% RSLogix 500 project LVD200820_BaseOnly_Mini.RSS, saved by version 11.00.00.00 %
PROJECT "LINL0619"    % processor: MicroLogix 1400 %

PROGRAM FILES
  LAD 2 "MAIN"  60 rungs  % Main Program Routine %
  LAD 4 "ENABLES"  16 rungs
  LAD 5 "FEED"  11 rungs  % normal %
  LAD 6 "SPEEDS"  12 rungs
  LAD 7 "HSC BOT"  5 rungs
  LAD 8 "HSC TOP"  5 rungs
  LAD 9 "1 MS STI"  22 rungs  % high speed %
  LAD 10 "SHIFT BOT"  8 rungs
  LAD 11 "SHIFT TOP"  10 rungs
  LAD 12 "BOTOPTIC"  3 rungs
  LAD 13 "BOTOPTMES"  7 rungs
  LAD 81 "I1"  1 rungs
  LAD 82 "I1 RESULT"  1 rungs
  LAD 83 "I1 PASS"  1 rungs
  LAD 84 "I1 FAIL"  1 rungs
  LAD 85 "I1 ACQ"  1 rungs
  LAD 86 "I1 TESTER"  1 rungs
  LAD 87 "I1 TRIG"  1 rungs
  LAD 88 "I1 FIFOSET"  1 rungs
  LAD 89 "I1 FIFOGET"  1 rungs
  LAD 90 "I1 DATA"  1 rungs
  LAD 91 "I1 FAULT"  1 rungs
  LAD 92 "I1 FIX1"  1 rungs
  LAD 93 "I1 FIX2"  1 rungs
  LAD 94 "I2"  1 rungs
  LAD 95 "I2 RESULT"  1 rungs
  LAD 96 "I2 PASS"  1 rungs
  LAD 97 "I2 FAIL"  1 rungs
  LAD 98 "I2 ACQ"  1 rungs
  LAD 99 "I2 TESTER"  1 rungs
  LAD 100 "I2 TRIG"  1 rungs
  LAD 101 "I2 FIFOSET"  1 rungs
  LAD 102 "I2 FIFOGET"  1 rungs
  LAD 103 "I2 DATA"  1 rungs
  LAD 104 "I2 FAULT"  1 rungs
  LAD 105 "I2 FIX1"  1 rungs
  LAD 106 "I2 FIX2"  1 rungs
  LAD 107 "I3"  1 rungs
  LAD 108 "I3 RESULT"  1 rungs
  LAD 109 "I3 PASS"  1 rungs
  LAD 110 "I3 FAIL"  1 rungs
  LAD 111 "I3 ACQ"  1 rungs
  LAD 112 "I3 TESTER"  1 rungs
  LAD 113 "I3 TRIG"  1 rungs
  LAD 114 "I3 FIFOSET"  1 rungs
  LAD 115 "I3 FIFOGET"  1 rungs
  LAD 116 "I3 DATA"  1 rungs
  LAD 117 "I3 FAULT"  1 rungs
  LAD 118 "I3 FIX1"  1 rungs
  LAD 119 "I3 FIX2"  1 rungs
  LAD 120 "I4"  1 rungs
  LAD 121 "I4 RESULT"  1 rungs
  LAD 122 "I4 PASS"  1 rungs
  LAD 123 "I4 FAIL"  1 rungs
  LAD 124 "I4 ACQ"  1 rungs
  LAD 125 "I4 TESTER"  1 rungs
  LAD 126 "I4 TRIG"  1 rungs
  LAD 127 "I4 FIFOSET"  1 rungs
  LAD 128 "I4 FIFOGET"  1 rungs
  LAD 129 "I4 DATA"  1 rungs
  LAD 130 "I4 FAULT"  1 rungs
  LAD 131 "I4 FIX1"  1 rungs
  LAD 132 "I4 FIX2"  1 rungs
  LAD 135 "XFER"  3 rungs
  LAD 137 "TOPOPTIC"  10 rungs
  LAD 138 "TOPOPVERT"  13 rungs
  LAD 139 "TOPOPREAL"  19 rungs
  LAD 140 "TOPOPTEST"  8 rungs
  LAD 141 "TOPOPRANGE"  6 rungs
  LAD 142 "TOPOPRANGE"  6 rungs
  LAD 143 "TOPOPOKAY"  6 rungs
  LAD 144 "TESTINJECT"  8 rungs
  LAD 148 "I5"  21 rungs
  LAD 149 "I5 RESULT"  7 rungs
  LAD 150 "I5 PASS"  6 rungs
  LAD 151 "I5 FAIL"  4 rungs
  LAD 152 "I5 ACQ"  9 rungs
  LAD 153 "I5 TESTER"  5 rungs
  LAD 154 "I5 TRIG"  5 rungs
  LAD 155 "I5 FIFOSET"  9 rungs
  LAD 156 "I5 FIFOGET"  8 rungs
  LAD 157 "I5 DATA"  3 rungs
  LAD 158 "I5 FAULT"  9 rungs
  LAD 159 "I5 FIX1"  5 rungs
  LAD 160 "I5 FIX2"  3 rungs
  LAD 161 "I6"  21 rungs
  LAD 162 "I6 RESULT"  7 rungs
  LAD 163 "I6 PASS"  5 rungs
  LAD 164 "I6 FAIL"  3 rungs
  LAD 165 "I6 ACQ"  8 rungs
  LAD 166 "I6 TESTER"  5 rungs
  LAD 167 "I6 TRIG"  5 rungs
  LAD 168 "I6 FIFOSET"  9 rungs
  LAD 169 "I6 FIFOGET"  8 rungs
  LAD 170 "I6 DATA"  3 rungs
  LAD 171 "I6 FAULT"  9 rungs
  LAD 172 "I6 FIX1"  5 rungs
  LAD 173 "I6 FIX2"  3 rungs
  LAD 174 "I7"  21 rungs
  LAD 175 "I7 RESULT"  7 rungs
  LAD 176 "I7 PASS"  6 rungs
  LAD 177 "I7 FAIL"  4 rungs
  LAD 178 "I7 ACQ"  9 rungs
  LAD 179 "I7 TESTER"  5 rungs
  LAD 180 "I7 TRIG"  5 rungs
  LAD 181 "I7 FIFOSET"  9 rungs
  LAD 182 "I7 FIFOGET"  8 rungs
  LAD 183 "I7 DATA"  3 rungs
  LAD 184 "I7 FAULT"  9 rungs
  LAD 185 "I7 FIX1"  5 rungs
  LAD 186 "I7 FIX2"  3 rungs
  LAD 187 "I8"  22 rungs
  LAD 188 "I8 RESULT"  7 rungs
  LAD 189 "I8 PASS"  6 rungs
  LAD 190 "I8 FAIL"  4 rungs
  LAD 191 "I8 ACQ"  9 rungs
  LAD 192 "I8 TESTER"  5 rungs
  LAD 193 "I8 TRIG"  5 rungs
  LAD 194 "I8 FIFOSET"  9 rungs
  LAD 195 "I8 FIFOGET"  8 rungs
  LAD 196 "I8 DATA"  3 rungs
  LAD 197 "I8 FAULT"  9 rungs
  LAD 198 "I8 FIX1"  5 rungs
  LAD 199 "I8 FIX2"  3 rungs
  LAD 200 "PASS BLOW"  15 rungs
  LAD 235 "TESTTRIGS"  7 rungs  % highspeed test triggers, not necessary %
  LAD 236 "TESTTRIG1"  4 rungs
  LAD 237 "TESTTRIG2"  4 rungs
  LAD 238 "TESTTRIG3"  4 rungs
  LAD 239 "TESTTRIG4"  4 rungs
  LAD 240 "TESTTRIG5"  4 rungs
  LAD 241 "TESTTRIG6"  4 rungs
  LAD 242 "TESTTRIG7"  4 rungs
  LAD 243 "TESTTRIG8"  4 rungs
  LAD 244 "PACKAGER"  28 rungs  % normal %
  LAD 245 "NO PACKAGE"  8 rungs
  LAD 246 "RATE1"  9 rungs
  LAD 247 "RATE2"  6 rungs
  LAD 248 "RESET RATE"  6 rungs
  LAD 249 "NP STOP"  8 rungs  % stop on no good %
  LAD 250 "SPEED BOT"  8 rungs  % high speed %
  LAD 251 "SPEED TOP"  8 rungs  % high speed %
  LAD 252 "P BOT"  7 rungs  % high speed %
  LAD 253 "P TOP"  7 rungs  % high speed %
  LAD 254 "TOTALCOUNT"  4 rungs
  LAD 255 "SAVED"  4 rungs

DATA FILES
  O0 OUTPUT  6 elements
  I1 INPUT  8 elements
  S2 STATUS  66 elements
  B3 BINARY  14 elements
  T4 TIMER  45 elements
  C5 COUNTER  1 elements
  R6 CONTROL  30 elements
  N7 INTEGER  200 elements
  F8 FLOAT  100 elements
  B12 HMI_BINARY  22 elements  % general use with hmi to avoid additional reads %
  L13  COUNTS  256 elements
  F14 HMI_FLOATS  100 elements
  N15 HMI_INTS  100 elements
  L16 HMI_LONGS  100 elements
  L19 RATE DATA  50 elements
  L20 I7TIMEFIFO  50 elements
  L21 I7POSFIFO  50 elements
  L22 I8TIMEFIFO  50 elements
  L23 I8POSFIFO  50 elements
  L30 INS5TIME  50 elements
  L31 INS5POS  50 elements
  L32 INS6TIME  50 elements
  L33 INS6POS  50 elements
  B34 BOT NG  128 elements
  B35 TOP NG  128 elements
  B36 BOTGOOD  128 elements
  B37 TOPGOOD1  128 elements
  B38 EX1 TEST  128 elements
  B39 TOPGOOD2  128 elements
  B40 EX2 TEST  128 elements
  N184 TEST INTS  50 elements
  L192 SPD OFFSET  50 elements
  B196 CTRL BITS  50 elements
  L199 USED  36 elements

LADDER 2 "MAIN"    % Main Program Routine %
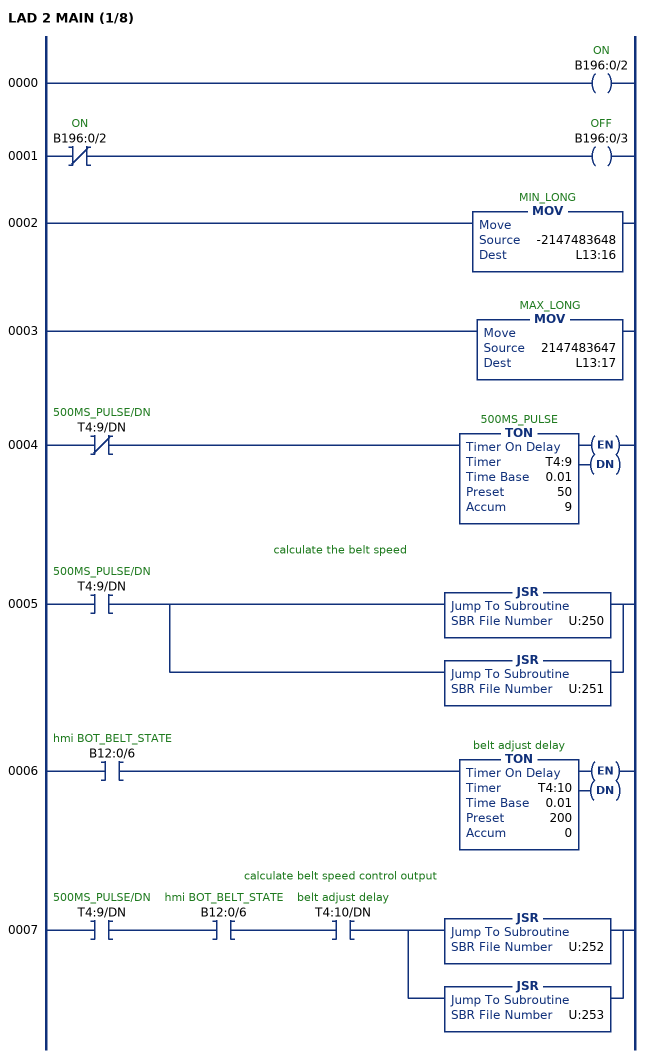
% Rung: 0 %
SOR OTE B196:0/2 EOR
%   B196:0/2  ON %
% Rung: 1 %
SOR XIO B196:0/2 OTE B196:0/3 EOR
%   B196:0/2  ON %
%   B196:0/3  OFF %
% Rung: 2 %
SOR MOV -2147483648 L13:16 EOR
%   L13:16  MIN_LONG %
% Rung: 3 %
SOR MOV 2147483647 L13:17 EOR
%   L13:17  MAX_LONG %
% Rung: 4 %
SOR XIO T4:9/DN TON T4:9 0.01 50 9 EOR
%   T4:9  500MS_PULSE %
% Rung: 5 %
% calculate the belt speed %
SOR XIC T4:9/DN BST JSR U:250 NXB JSR U:251 BND EOR
%   T4:9  500MS_PULSE %
% Rung: 6 %
SOR XIC B12:0/6 TON T4:10 0.01 200 0 EOR
%   B12:0/6  BOT_BELT_STATE  "hmi" %
%   T4:10  "belt adjust delay" %
% Rung: 7 %
% calculate belt speed control output %
SOR XIC T4:9/DN XIC B12:0/6 XIC T4:10/DN BST JSR U:252 NXB JSR U:253 BND EOR
%   T4:9  500MS_PULSE %
%   B12:0/6  BOT_BELT_STATE  "hmi" %
%   T4:10  "belt adjust delay" %

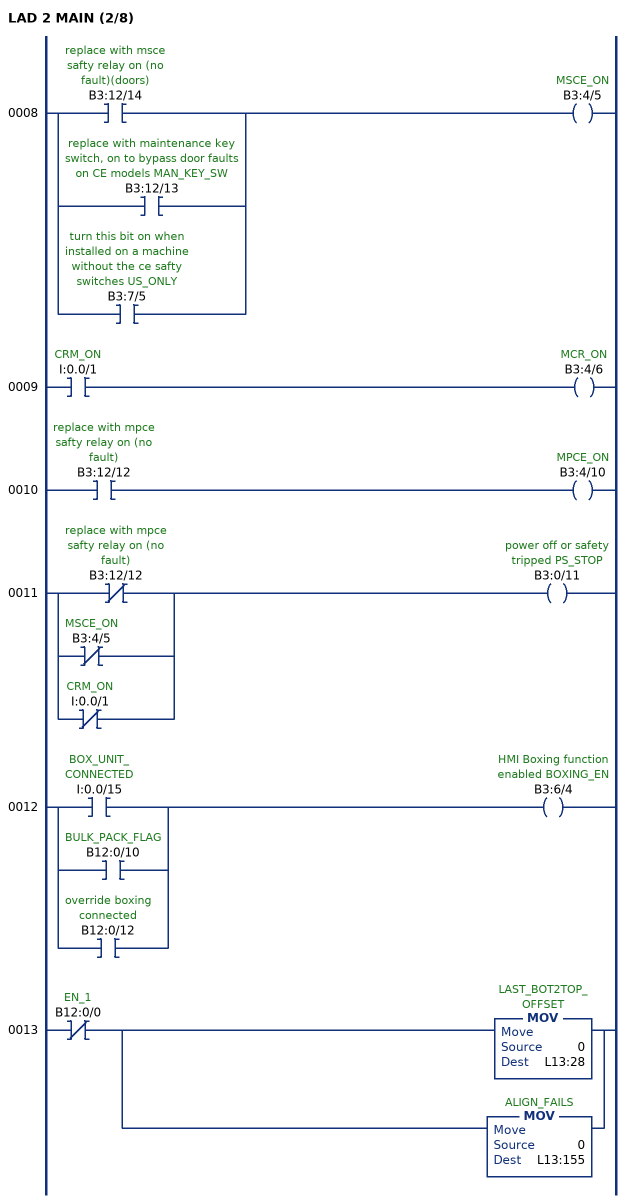
% Rung: 8 %
SOR BST XIC B3:12/14 NXB XIC B3:12/13 NXB XIC B3:7/5 BND OTE B3:4/5 EOR
%   B3:12/14  "replace with msce safty relay on (no fault)(doors)" %
%   B3:12/13  MAN_KEY_SW  "replace with maintenance key switch, on to bypass door faults on CE models" %
%   B3:7/5  US_ONLY  "turn this bit on when installed on a machine without the ce safty switches" %
%   B3:4/5  MSCE_ON %
% Rung: 9 %
SOR XIC I:0.0/1 OTE B3:4/6 EOR
%   I:0.0/1  CRM_ON %
%   B3:4/6  MCR_ON %
% Rung: 10 %
SOR XIC B3:12/12 OTE B3:4/10 EOR
%   B3:12/12  "replace with mpce safty relay on (no fault)" %
%   B3:4/10  MPCE_ON %
% Rung: 11 %
SOR BST XIO B3:12/12 NXB XIO B3:4/5 NXB XIO I:0.0/1 BND OTE B3:0/11 EOR
%   B3:12/12  "replace with mpce safty relay on (no fault)" %
%   B3:4/5  MSCE_ON %
%   I:0.0/1  CRM_ON %
%   B3:0/11  PS_STOP  "power off or safety tripped" %
% Rung: 12 %
SOR BST XIC I:0.0/15 NXB XIC B12:0/10 NXB XIC B12:0/12 BND OTE B3:6/4 EOR
%   I:0.0/15  BOX_UNIT_CONNECTED %
%   B12:0/10  BULK_PACK_FLAG %
%   B12:0/12  "override boxing connected" %
%   B3:6/4  BOXING_EN  "HMI Boxing function enabled" %
% Rung: 13 %
SOR XIO B12:0/0 BST MOV 0 L13:28 NXB MOV 0 L13:155 BND EOR
%   B12:0/0  EN_1 %
%   L13:28  LAST_BOT2TOP_OFFSET %
%   L13:155  ALIGN_FAILS %

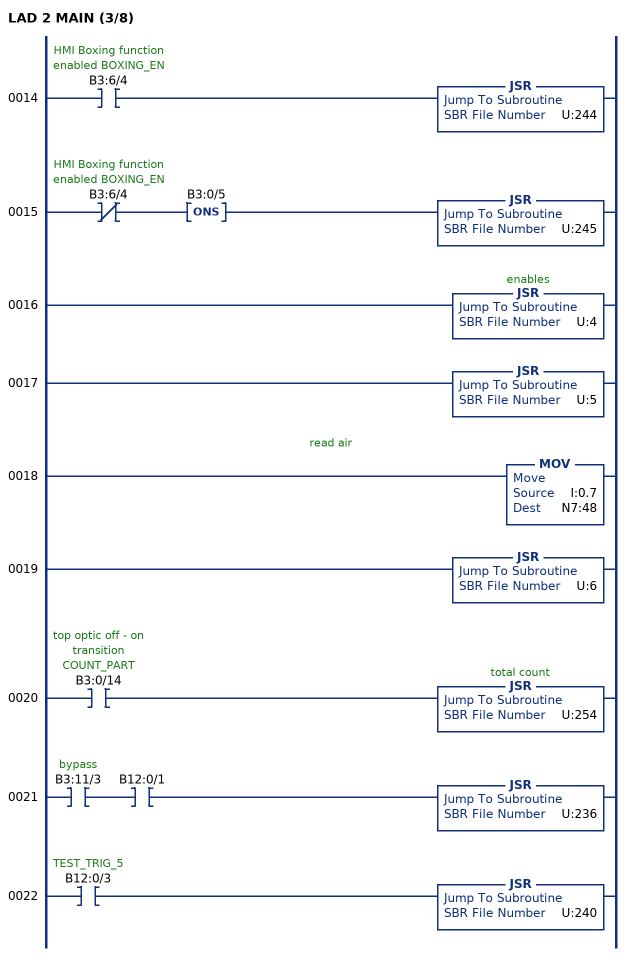
% Rung: 14 %
SOR XIC B3:6/4 JSR U:244 EOR
%   B3:6/4  BOXING_EN  "HMI Boxing function enabled" %
% Rung: 15 %
SOR XIO B3:6/4 ONS B3:0/5 JSR U:245 EOR
%   B3:6/4  BOXING_EN  "HMI Boxing function enabled" %
% Rung: 16 %
SOR JSR U:4 EOR
%   U:4  "enables" %
% Rung: 17 %
SOR JSR U:5 EOR
% Rung: 18 %
% read air %
SOR MOV I:0.7 N7:48 EOR
%   I:0.7  "Air Presure Sensor Input Signal" %
% Rung: 19 %
SOR JSR U:6 EOR
% Rung: 20 %
SOR XIC B3:0/14 JSR U:254 EOR
%   B3:0/14  COUNT_PART  "top optic off - on transition" %
%   U:254  "total count" %
% Rung: 21 %
SOR XIC B3:11/3 XIC B12:0/1 JSR U:236 EOR
%   B3:11/3  "bypass" %
% Rung: 22 %
SOR XIC B12:0/3 JSR U:240 EOR
%   B12:0/3  TEST_TRIG_5 %

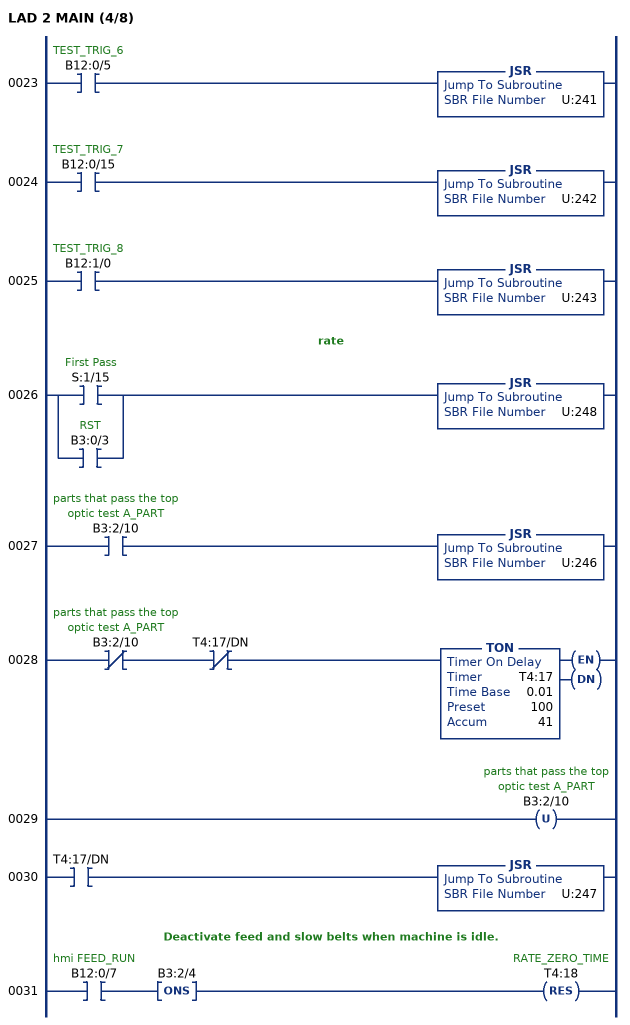
% Rung: 23 %
SOR XIC B12:0/5 JSR U:241 EOR
%   B12:0/5  TEST_TRIG_6 %
% Rung: 24 %
SOR XIC B12:0/15 JSR U:242 EOR
%   B12:0/15  TEST_TRIG_7 %
% Rung: 25 %
SOR XIC B12:1/0 JSR U:243 EOR
%   B12:1/0  TEST_TRIG_8 %
% Rung: 26 %
% TITLE: rate %
SOR BST XIC S:1/15 NXB XIC B3:0/3 BND JSR U:248 EOR
%   S:1/15  "First Pass" %
%   B3:0/3  RST %
% Rung: 27 %
SOR XIC B3:2/10 JSR U:246 EOR
%   B3:2/10  A_PART  "parts that pass the top optic test" %
% Rung: 28 %
SOR XIO B3:2/10 XIO T4:17/DN TON T4:17 0.01 100 41 EOR
%   B3:2/10  A_PART  "parts that pass the top optic test" %
% Rung: 29 %
SOR OTU B3:2/10 EOR
%   B3:2/10  A_PART  "parts that pass the top optic test" %
% Rung: 30 %
SOR XIC T4:17/DN JSR U:247 EOR
% Rung: 31 %
% TITLE: Deactivate feed and slow belts when machine is idle. %
SOR XIC B12:0/7 ONS B3:2/4 RES T4:18 EOR
%   B12:0/7  FEED_RUN  "hmi" %
%   T4:18  RATE_ZERO_TIME %

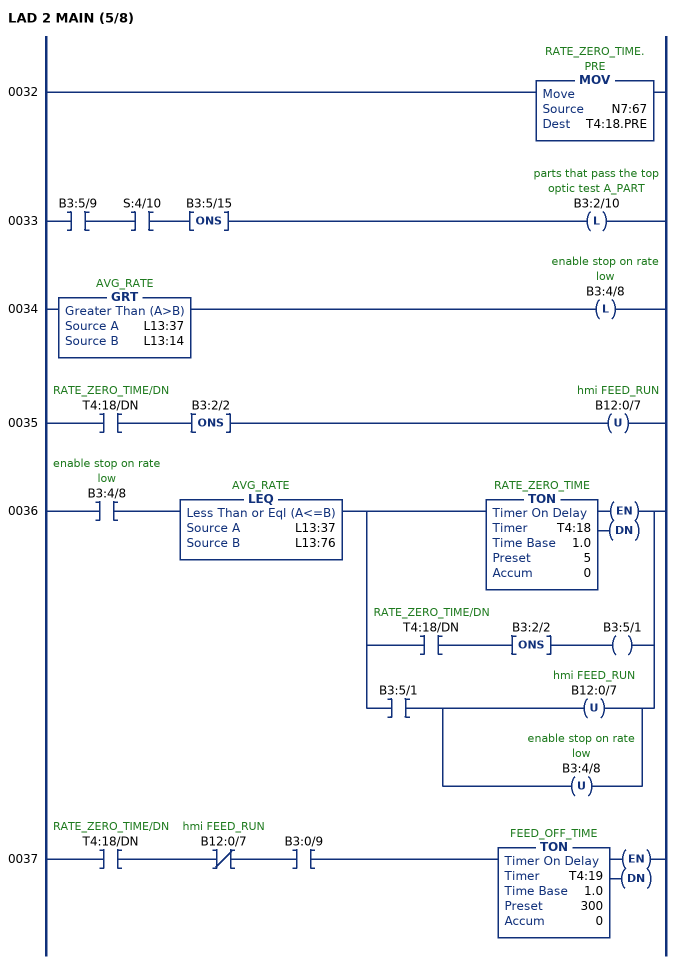
% Rung: 32 %
SOR MOV N7:67 T4:18.PRE EOR
%   N7:67  "empty bowl or jam bowl run time" %
%   T4:18  RATE_ZERO_TIME %
% Rung: 33 %
SOR XIC B3:5/9 XIC S:4/10 ONS B3:5/15 OTL B3:2/10 EOR
%   B3:2/10  A_PART  "parts that pass the top optic test" %
% Rung: 34 %
SOR GRT L13:37 L13:14 OTL B3:4/8 EOR
%   L13:37  AVG_RATE %
%   B3:4/8  "enable stop on rate low" %
% Rung: 35 %
SOR XIC T4:18/DN ONS B3:2/2 OTU B12:0/7 EOR
%   T4:18  RATE_ZERO_TIME %
%   B12:0/7  FEED_RUN  "hmi" %
% Rung: 36 %
SOR XIC B3:4/8 LEQ L13:37 L13:76 BST TON T4:18 1.0 5 0 NXB XIC T4:18/DN ONS B3:2/2 OTE B3:5/1 NXB XIC B3:5/1 BST OTU B12:0/7 NXB OTU B3:4/8 BND BND EOR
%   B3:4/8  "enable stop on rate low" %
%   L13:37  AVG_RATE %
%   T4:18  RATE_ZERO_TIME %
%   B12:0/7  FEED_RUN  "hmi" %
% Rung: 37 %
SOR XIC T4:18/DN XIO B12:0/7 XIC B3:0/9 TON T4:19 1.0 300 0 EOR
%   T4:18  RATE_ZERO_TIME %
%   B12:0/7  FEED_RUN  "hmi" %
%   T4:19  FEED_OFF_TIME %

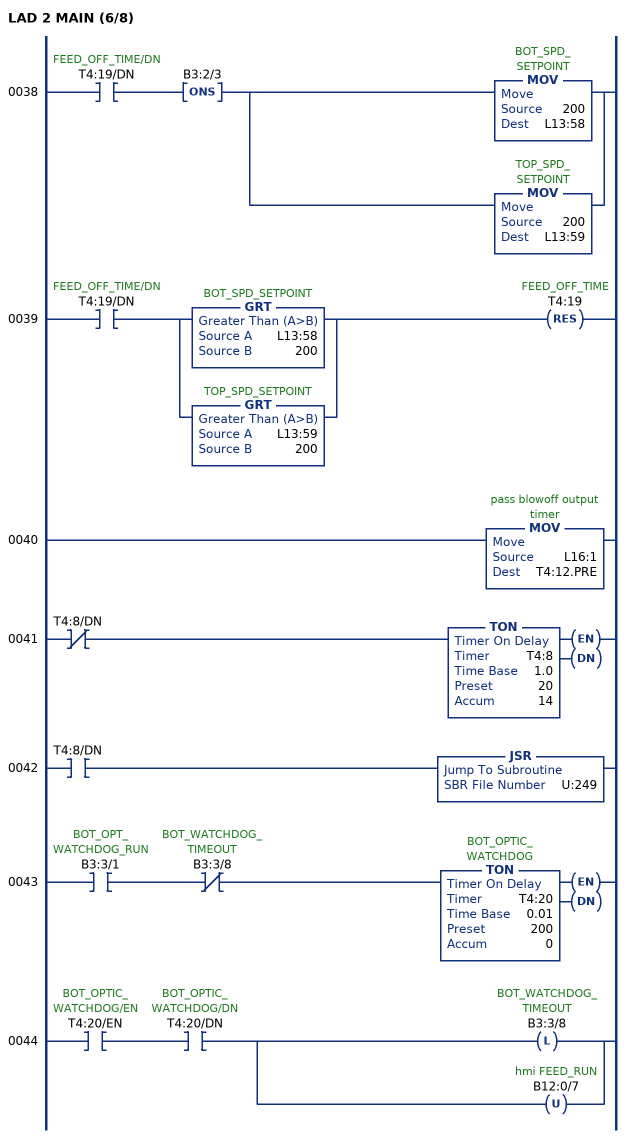
% Rung: 38 %
SOR XIC T4:19/DN ONS B3:2/3 BST MOV 200 L13:58 NXB MOV 200 L13:59 BND EOR
%   T4:19  FEED_OFF_TIME %
%   L13:58  BOT_SPD_SETPOINT %
%   L13:59  TOP_SPD_SETPOINT %
% Rung: 39 %
SOR XIC T4:19/DN BST GRT L13:58 200 NXB GRT L13:59 200 BND RES T4:19 EOR
%   T4:19  FEED_OFF_TIME %
%   L13:58  BOT_SPD_SETPOINT %
%   L13:59  TOP_SPD_SETPOINT %
% Rung: 40 %
SOR MOV L16:1 T4:12.PRE EOR
%   L16:1  BLOW_TIME %
%   T4:12  "pass blowoff output timer" %
% Rung: 41 %
SOR XIO T4:8/DN TON T4:8 1.0 20 14 EOR
% Rung: 42 %
SOR XIC T4:8/DN JSR U:249 EOR
% Rung: 43 %
SOR XIC B3:3/1 XIO B3:3/8 TON T4:20 0.01 200 0 EOR
%   B3:3/1  BOT_OPT_WATCHDOG_RUN %
%   B3:3/8  BOT_WATCHDOG_TIMEOUT %
%   T4:20  BOT_OPTIC_WATCHDOG %
% Rung: 44 %
SOR XIC T4:20/EN XIC T4:20/DN BST OTL B3:3/8 NXB OTU B12:0/7 BND EOR
%   T4:20  BOT_OPTIC_WATCHDOG %
%   B3:3/8  BOT_WATCHDOG_TIMEOUT %
%   B12:0/7  FEED_RUN  "hmi" %

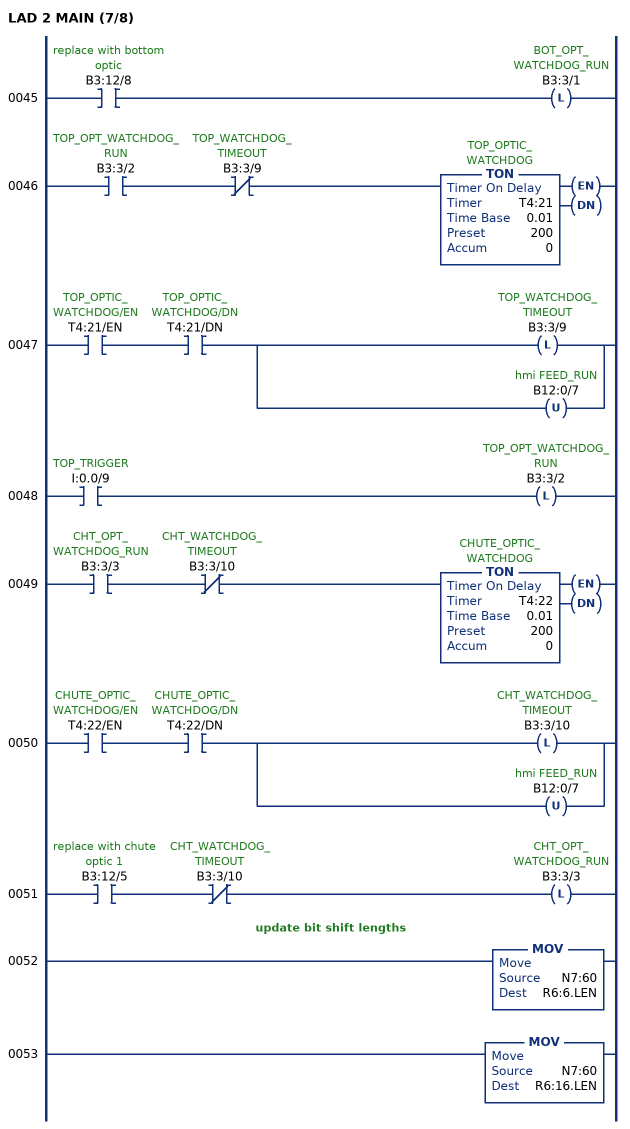
% Rung: 45 %
SOR XIC B3:12/8 OTL B3:3/1 EOR
%   B3:12/8  "replace with bottom optic" %
%   B3:3/1  BOT_OPT_WATCHDOG_RUN %
% Rung: 46 %
SOR XIC B3:3/2 XIO B3:3/9 TON T4:21 0.01 200 0 EOR
%   B3:3/2  TOP_OPT_WATCHDOG_RUN %
%   B3:3/9  TOP_WATCHDOG_TIMEOUT %
%   T4:21  TOP_OPTIC_WATCHDOG %
% Rung: 47 %
SOR XIC T4:21/EN XIC T4:21/DN BST OTL B3:3/9 NXB OTU B12:0/7 BND EOR
%   T4:21  TOP_OPTIC_WATCHDOG %
%   B3:3/9  TOP_WATCHDOG_TIMEOUT %
%   B12:0/7  FEED_RUN  "hmi" %
% Rung: 48 %
SOR XIC I:0.0/9 OTL B3:3/2 EOR
%   I:0.0/9  TOP_TRIGGER %
%   B3:3/2  TOP_OPT_WATCHDOG_RUN %
% Rung: 49 %
SOR XIC B3:3/3 XIO B3:3/10 TON T4:22 0.01 200 0 EOR
%   B3:3/3  CHT_OPT_WATCHDOG_RUN %
%   B3:3/10  CHT_WATCHDOG_TIMEOUT %
%   T4:22  CHUTE_OPTIC_WATCHDOG %
% Rung: 50 %
SOR XIC T4:22/EN XIC T4:22/DN BST OTL B3:3/10 NXB OTU B12:0/7 BND EOR
%   T4:22  CHUTE_OPTIC_WATCHDOG %
%   B3:3/10  CHT_WATCHDOG_TIMEOUT %
%   B12:0/7  FEED_RUN  "hmi" %
% Rung: 51 %
SOR XIC B3:12/5 XIO B3:3/10 OTL B3:3/3 EOR
%   B3:12/5  "replace with chute optic 1" %
%   B3:3/10  CHT_WATCHDOG_TIMEOUT %
%   B3:3/3  CHT_OPT_WATCHDOG_RUN %
% Rung: 52 %
% TITLE: update bit shift lengths %
SOR MOV N7:60 R6:6.LEN EOR
% Rung: 53 %
SOR MOV N7:60 R6:16.LEN EOR

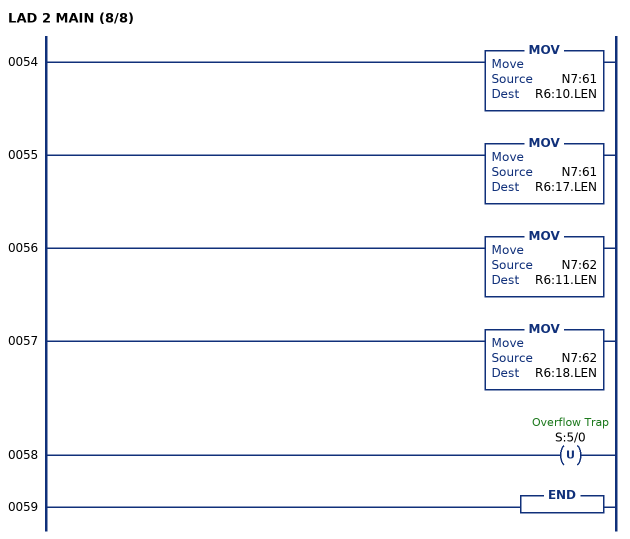
% Rung: 54 %
SOR MOV N7:61 R6:10.LEN EOR
% Rung: 55 %
SOR MOV N7:61 R6:17.LEN EOR
% Rung: 56 %
SOR MOV N7:62 R6:11.LEN EOR
% Rung: 57 %
SOR MOV N7:62 R6:18.LEN EOR
% Rung: 58 %
SOR OTU S:5/0 EOR
%   S:5/0  "Overflow Trap" %
% Rung: 59 %
SOR END EOR

LADDER 4 "ENABLES"
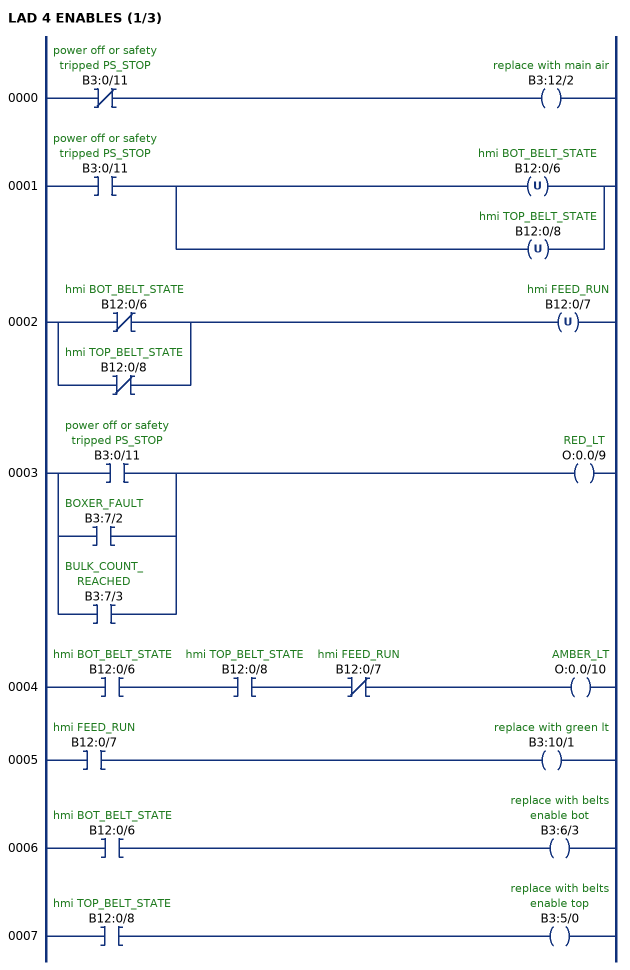
% Rung: 0 %
SOR XIO B3:0/11 OTE B3:12/2 EOR
%   B3:0/11  PS_STOP  "power off or safety tripped" %
%   B3:12/2  "replace with main air" %
% Rung: 1 %
SOR XIC B3:0/11 BST OTU B12:0/6 NXB OTU B12:0/8 BND EOR
%   B3:0/11  PS_STOP  "power off or safety tripped" %
%   B12:0/6  BOT_BELT_STATE  "hmi" %
%   B12:0/8  TOP_BELT_STATE  "hmi" %
% Rung: 2 %
SOR BST XIO B12:0/6 NXB XIO B12:0/8 BND OTU B12:0/7 EOR
%   B12:0/6  BOT_BELT_STATE  "hmi" %
%   B12:0/8  TOP_BELT_STATE  "hmi" %
%   B12:0/7  FEED_RUN  "hmi" %
% Rung: 3 %
SOR BST XIC B3:0/11 NXB XIC B3:7/2 NXB XIC B3:7/3 BND OTE O:0.0/9 EOR
%   B3:0/11  PS_STOP  "power off or safety tripped" %
%   B3:7/2  BOXER_FAULT %
%   B3:7/3  BULK_COUNT_REACHED %
%   O:0.0/9  RED_LT %
% Rung: 4 %
SOR XIC B12:0/6 XIC B12:0/8 XIO B12:0/7 OTE O:0.0/10 EOR
%   B12:0/6  BOT_BELT_STATE  "hmi" %
%   B12:0/8  TOP_BELT_STATE  "hmi" %
%   B12:0/7  FEED_RUN  "hmi" %
%   O:0.0/10  AMBER_LT %
% Rung: 5 %
SOR XIC B12:0/7 OTE B3:10/1 EOR
%   B12:0/7  FEED_RUN  "hmi" %
%   B3:10/1  "replace with green lt" %
% Rung: 6 %
SOR XIC B12:0/6 OTE B3:6/3 EOR
%   B12:0/6  BOT_BELT_STATE  "hmi" %
%   B3:6/3  "replace with belts enable bot" %
% Rung: 7 %
SOR XIC B12:0/8 OTE B3:5/0 EOR
%   B12:0/8  TOP_BELT_STATE  "hmi" %
%   B3:5/0  "replace with belts enable top" %

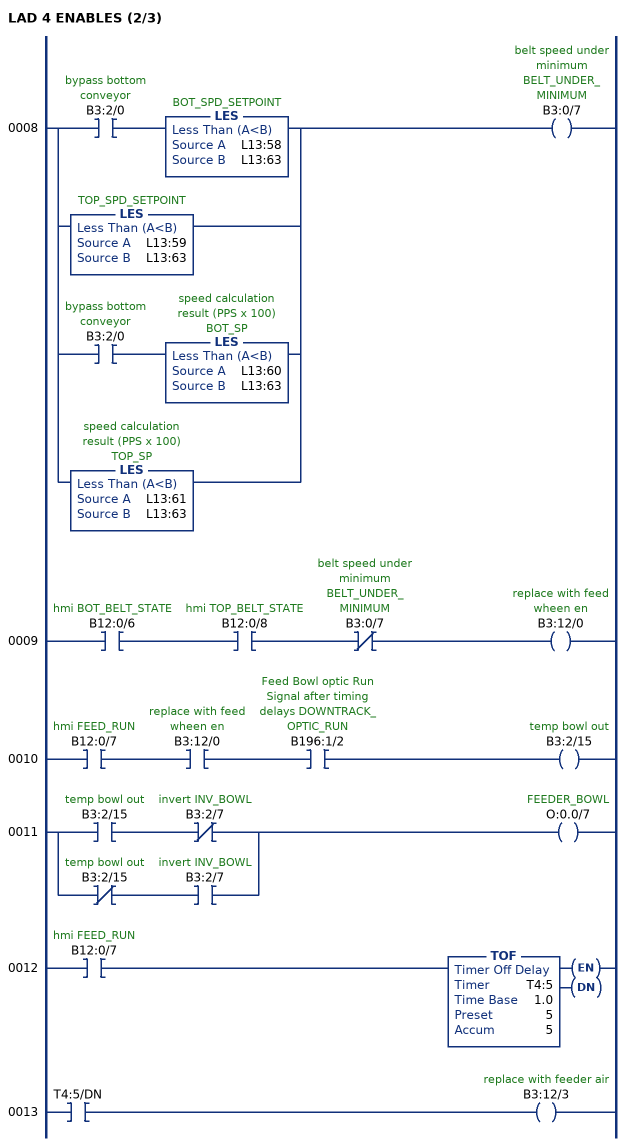
% Rung: 8 %
SOR BST XIC B3:2/0 LES L13:58 L13:63 NXB LES L13:59 L13:63 NXB XIC B3:2/0 LES L13:60 L13:63 NXB LES L13:61 L13:63 BND OTE B3:0/7 EOR
%   B3:2/0  "bypass bottom conveyor" %
%   L13:58  BOT_SPD_SETPOINT %
%   L13:63  "min belt speed" %
%   L13:59  TOP_SPD_SETPOINT %
%   L13:60  BOT_SP  "speed calculation result (PPS x 100)" %
%   L13:61  TOP_SP  "speed calculation result (PPS x 100)" %
%   B3:0/7  BELT_UNDER_MINIMUM  "belt speed under minimum" %
% Rung: 9 %
SOR XIC B12:0/6 XIC B12:0/8 XIO B3:0/7 OTE B3:12/0 EOR
%   B12:0/6  BOT_BELT_STATE  "hmi" %
%   B12:0/8  TOP_BELT_STATE  "hmi" %
%   B3:0/7  BELT_UNDER_MINIMUM  "belt speed under minimum" %
%   B3:12/0  "replace with feed wheen en" %
% Rung: 10 %
SOR XIC B12:0/7 XIC B3:12/0 XIC B196:1/2 OTE B3:2/15 EOR
%   B12:0/7  FEED_RUN  "hmi" %
%   B3:12/0  "replace with feed wheen en" %
%   B196:1/2  DOWNTRACK_OPTIC_RUN  "Feed Bowl optic Run Signal after timing delays" %
%   B3:2/15  "temp bowl out" %
% Rung: 11 %
SOR BST XIC B3:2/15 XIO B3:2/7 NXB XIO B3:2/15 XIC B3:2/7 BND OTE O:0.0/7 EOR
%   B3:2/15  "temp bowl out" %
%   B3:2/7  INV_BOWL  "invert" %
%   O:0.0/7  FEEDER_BOWL %
% Rung: 12 %
SOR XIC B12:0/7 TOF T4:5 1.0 5 5 EOR
%   B12:0/7  FEED_RUN  "hmi" %
% Rung: 13 %
SOR XIC T4:5/DN OTE B3:12/3 EOR
%   B3:12/3  "replace with feeder air" %

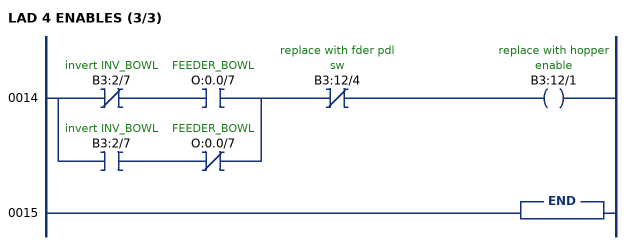
% Rung: 14 %
SOR BST XIO B3:2/7 XIC O:0.0/7 NXB XIC B3:2/7 XIO O:0.0/7 BND XIO B3:12/4 OTE B3:12/1 EOR
%   B3:2/7  INV_BOWL  "invert" %
%   O:0.0/7  FEEDER_BOWL %
%   B3:12/4  "replace with fder pdl sw" %
%   B3:12/1  "replace with hopper enable" %
% Rung: 15 %
SOR END EOR

LADDER 5 "FEED"    % normal %
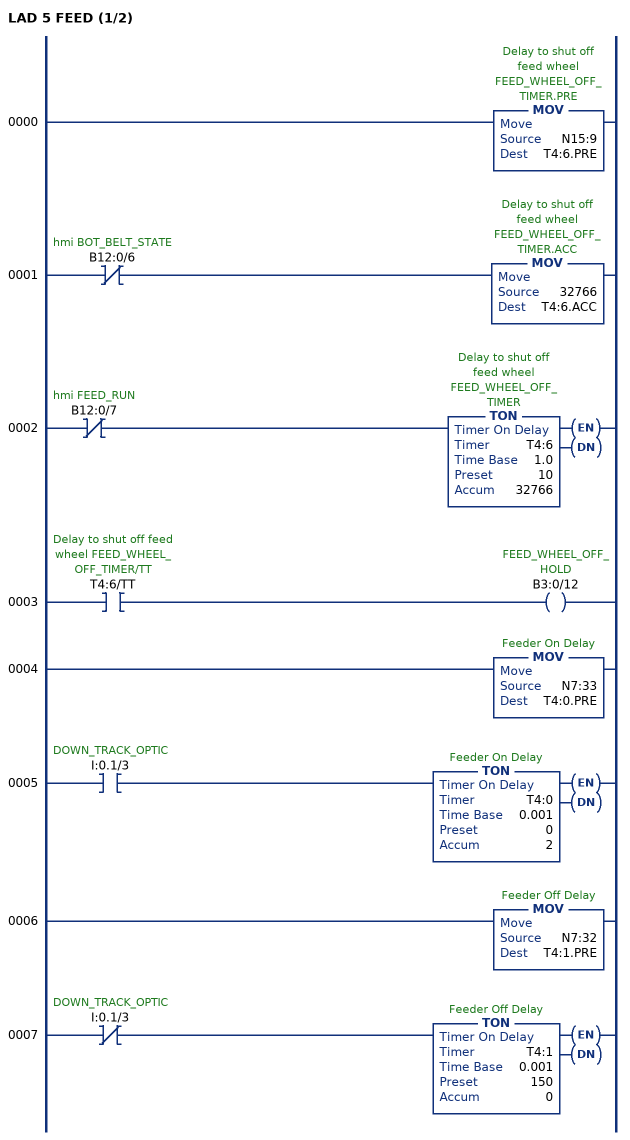
% Rung: 0 %
SOR MOV N15:9 T4:6.PRE EOR
%   N15:9  FEED_WHEEL_STOP_TIME %
%   T4:6  FEED_WHEEL_OFF_TIMER  "Delay to shut off feed wheel" %
% Rung: 1 %
SOR XIO B12:0/6 MOV 32766 T4:6.ACC EOR
%   B12:0/6  BOT_BELT_STATE  "hmi" %
%   T4:6  FEED_WHEEL_OFF_TIMER  "Delay to shut off feed wheel" %
% Rung: 2 %
SOR XIO B12:0/7 TON T4:6 1.0 10 32766 EOR
%   B12:0/7  FEED_RUN  "hmi" %
%   T4:6  FEED_WHEEL_OFF_TIMER  "Delay to shut off feed wheel" %
% Rung: 3 %
SOR XIC T4:6/TT OTE B3:0/12 EOR
%   T4:6  FEED_WHEEL_OFF_TIMER  "Delay to shut off feed wheel" %
%   B3:0/12  FEED_WHEEL_OFF_HOLD %
% Rung: 4 %
SOR MOV N7:33 T4:0.PRE EOR
%   N7:33  "down track on delay" %
%   T4:0  "Feeder On Delay" %
% Rung: 5 %
SOR XIC I:0.1/3 TON T4:0 0.001 0 2 EOR
%   I:0.1/3  DOWN_TRACK_OPTIC %
%   T4:0  "Feeder On Delay" %
% Rung: 6 %
SOR MOV N7:32 T4:1.PRE EOR
%   N7:32  "down track off delay" %
%   T4:1  "Feeder Off Delay" %
% Rung: 7 %
SOR XIO I:0.1/3 TON T4:1 0.001 150 0 EOR
%   I:0.1/3  DOWN_TRACK_OPTIC %
%   T4:1  "Feeder Off Delay" %

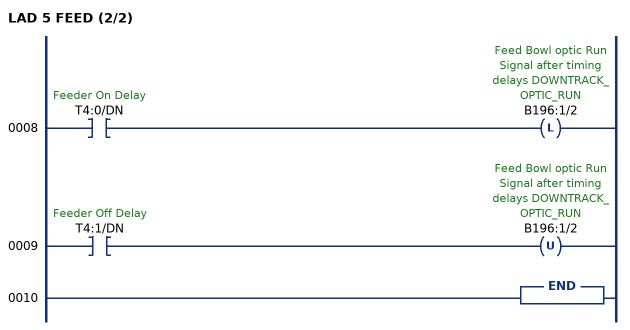
% Rung: 8 %
SOR XIC T4:0/DN OTL B196:1/2 EOR
%   T4:0  "Feeder On Delay" %
%   B196:1/2  DOWNTRACK_OPTIC_RUN  "Feed Bowl optic Run Signal after timing delays" %
% Rung: 9 %
SOR XIC T4:1/DN OTU B196:1/2 EOR
%   T4:1  "Feeder Off Delay" %
%   B196:1/2  DOWNTRACK_OPTIC_RUN  "Feed Bowl optic Run Signal after timing delays" %
% Rung: 10 %
SOR END EOR

LADDER 6 "SPEEDS"
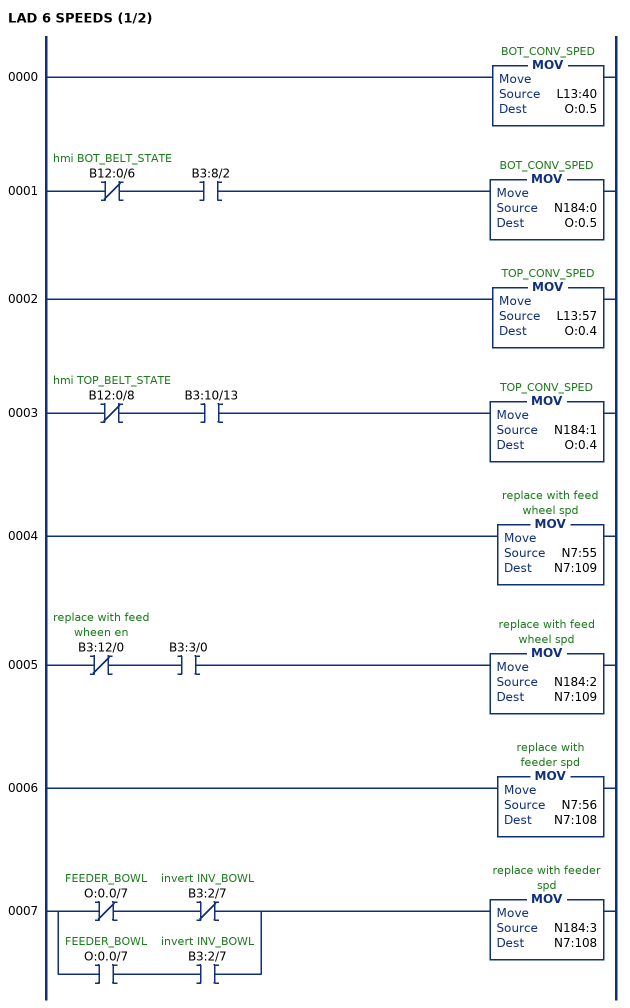
% Rung: 0 %
SOR MOV L13:40 O:0.5 EOR
%   L13:40  SCALED_BOT_VALUE %
%   O:0.5  BOT_CONV_SPED %
% Rung: 1 %
SOR XIO B12:0/6 XIC B3:8/2 MOV N184:0 O:0.5 EOR
%   B12:0/6  BOT_BELT_STATE  "hmi" %
%   O:0.5  BOT_CONV_SPED %
% Rung: 2 %
SOR MOV L13:57 O:0.4 EOR
%   L13:57  SCALED_TOP_VALUE %
%   O:0.4  TOP_CONV_SPED %
% Rung: 3 %
SOR XIO B12:0/8 XIC B3:10/13 MOV N184:1 O:0.4 EOR
%   B12:0/8  TOP_BELT_STATE  "hmi" %
%   O:0.4  TOP_CONV_SPED %
% Rung: 4 %
SOR MOV N7:55 N7:109 EOR
%   N7:109  "replace with feed wheel spd" %
% Rung: 5 %
SOR XIO B3:12/0 XIC B3:3/0 MOV N184:2 N7:109 EOR
%   B3:12/0  "replace with feed wheen en" %
%   N7:109  "replace with feed wheel spd" %
% Rung: 6 %
SOR MOV N7:56 N7:108 EOR
%   N7:108  "replace with feeder spd" %
% Rung: 7 %
SOR BST XIO O:0.0/7 XIO B3:2/7 NXB XIC O:0.0/7 XIC B3:2/7 BND MOV N184:3 N7:108 EOR
%   O:0.0/7  FEEDER_BOWL %
%   B3:2/7  INV_BOWL  "invert" %
%   N7:108  "replace with feeder spd" %

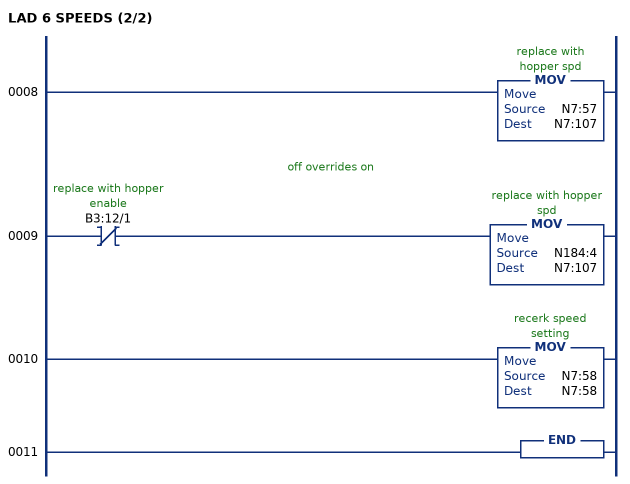
% Rung: 8 %
SOR MOV N7:57 N7:107 EOR
%   N7:107  "replace with hopper spd" %
% Rung: 9 %
% off overrides on %
SOR XIO B3:12/1 MOV N184:4 N7:107 EOR
%   B3:12/1  "replace with hopper enable" %
%   N7:107  "replace with hopper spd" %
% Rung: 10 %
SOR MOV N7:58 N7:58 EOR
%   N7:58  "recerk speed setting" %
% Rung: 11 %
SOR END EOR

LADDER 7 "HSC BOT"
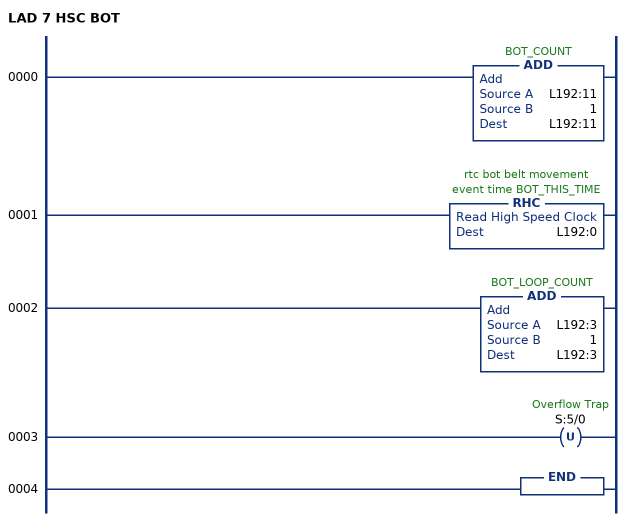
% Rung: 0 %
SOR ADD L192:11 1 L192:11 EOR
%   L192:11  BOT_COUNT %
% Rung: 1 %
SOR RHC L192:0 EOR
%   L192:0  BOT_THIS_TIME  "rtc bot belt movement event time" %
% Rung: 2 %
SOR ADD L192:3 1 L192:3 EOR
%   L192:3  BOT_LOOP_COUNT %
% Rung: 3 %
SOR OTU S:5/0 EOR
%   S:5/0  "Overflow Trap" %
% Rung: 4 %
SOR END EOR

LADDER 8 "HSC TOP"
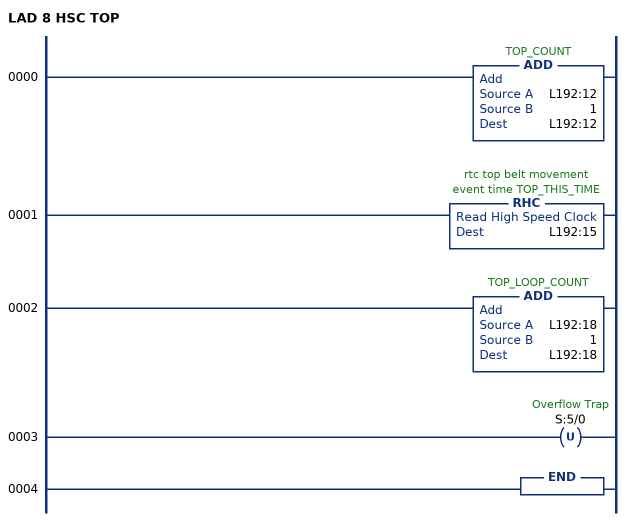
% Rung: 0 %
SOR ADD L192:12 1 L192:12 EOR
%   L192:12  TOP_COUNT %
% Rung: 1 %
SOR RHC L192:15 EOR
%   L192:15  TOP_THIS_TIME  "rtc top belt movement event time" %
% Rung: 2 %
SOR ADD L192:18 1 L192:18 EOR
%   L192:18  TOP_LOOP_COUNT %
% Rung: 3 %
SOR OTU S:5/0 EOR
%   S:5/0  "Overflow Trap" %
% Rung: 4 %
SOR END EOR

LADDER 9 "1 MS STI"    % high speed %
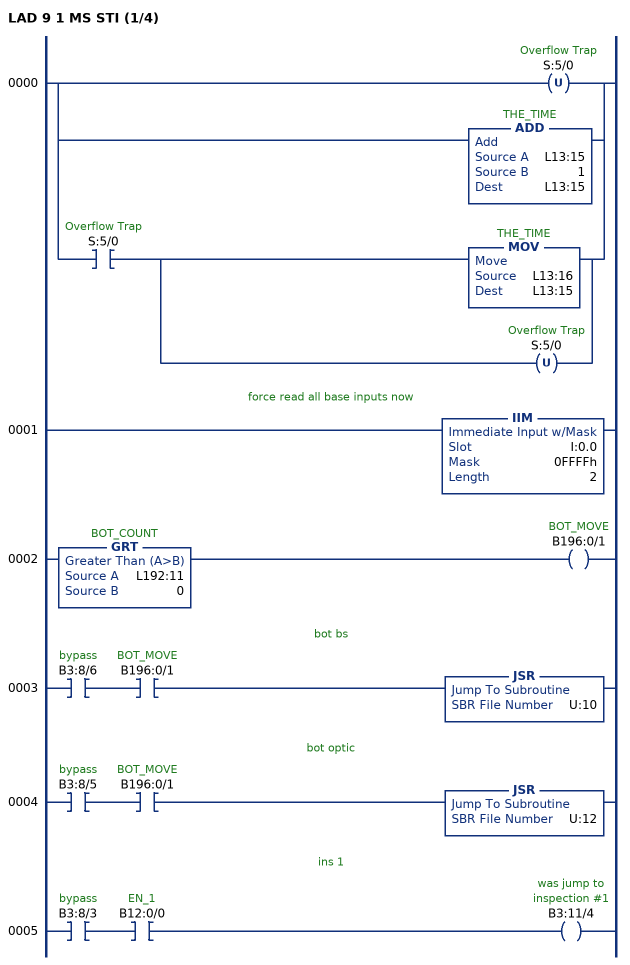
% Rung: 0 %
SOR BST OTU S:5/0 NXB ADD L13:15 1 L13:15 NXB XIC S:5/0 BST MOV L13:16 L13:15 NXB OTU S:5/0 BND BND EOR
%   S:5/0  "Overflow Trap" %
%   L13:15  THE_TIME %
%   L13:16  MIN_LONG %
% Rung: 1 %
% force read all base inputs now %
SOR IIM I:0.0 0FFFFh 2 EOR
% Rung: 2 %
SOR GRT L192:11 0 OTE B196:0/1 EOR
%   L192:11  BOT_COUNT %
%   B196:0/1  BOT_MOVE %
% Rung: 3 %
% bot bs %
SOR XIC B3:8/6 XIC B196:0/1 JSR U:10 EOR
%   B3:8/6  "bypass" %
%   B196:0/1  BOT_MOVE %
% Rung: 4 %
% bot optic %
SOR XIC B3:8/5 XIC B196:0/1 JSR U:12 EOR
%   B3:8/5  "bypass" %
%   B196:0/1  BOT_MOVE %
% Rung: 5 %
% ins 1 %
SOR XIC B3:8/3 XIC B12:0/0 OTE B3:11/4 EOR
%   B3:8/3  "bypass" %
%   B12:0/0  EN_1 %
%   B3:11/4  "was jump to inspection #1" %

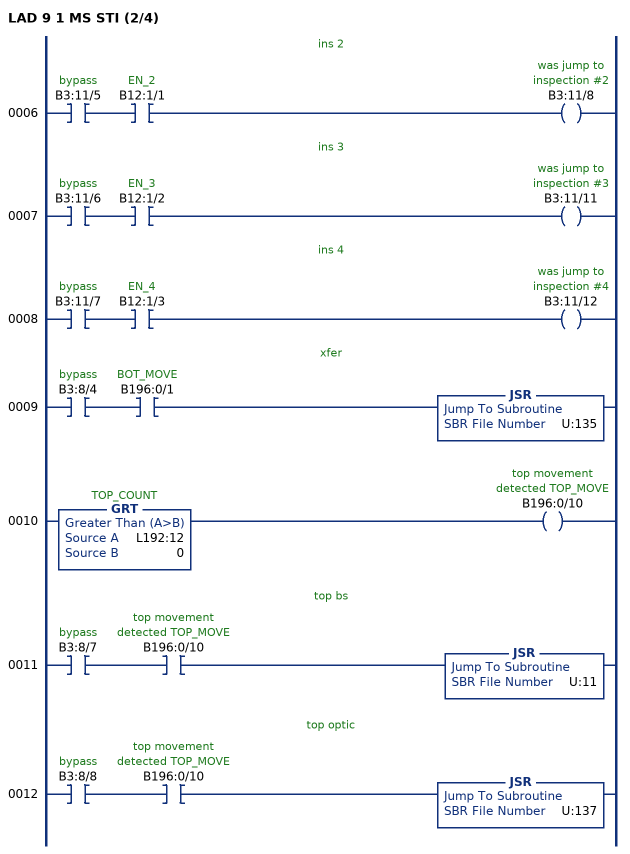
% Rung: 6 %
% ins 2 %
SOR XIC B3:11/5 XIC B12:1/1 OTE B3:11/8 EOR
%   B3:11/5  "bypass" %
%   B12:1/1  EN_2 %
%   B3:11/8  "was jump to inspection #2" %
% Rung: 7 %
% ins 3 %
SOR XIC B3:11/6 XIC B12:1/2 OTE B3:11/11 EOR
%   B3:11/6  "bypass" %
%   B12:1/2  EN_3 %
%   B3:11/11  "was jump to inspection #3" %
% Rung: 8 %
% ins 4 %
SOR XIC B3:11/7 XIC B12:1/3 OTE B3:11/12 EOR
%   B3:11/7  "bypass" %
%   B12:1/3  EN_4 %
%   B3:11/12  "was jump to inspection #4" %
% Rung: 9 %
% xfer %
SOR XIC B3:8/4 XIC B196:0/1 JSR U:135 EOR
%   B3:8/4  "bypass" %
%   B196:0/1  BOT_MOVE %
% Rung: 10 %
SOR GRT L192:12 0 OTE B196:0/10 EOR
%   L192:12  TOP_COUNT %
%   B196:0/10  TOP_MOVE  "top movement detected" %
% Rung: 11 %
% top bs %
SOR XIC B3:8/7 XIC B196:0/10 JSR U:11 EOR
%   B3:8/7  "bypass" %
%   B196:0/10  TOP_MOVE  "top movement detected" %
% Rung: 12 %
% top optic %
SOR XIC B3:8/8 XIC B196:0/10 JSR U:137 EOR
%   B3:8/8  "bypass" %
%   B196:0/10  TOP_MOVE  "top movement detected" %

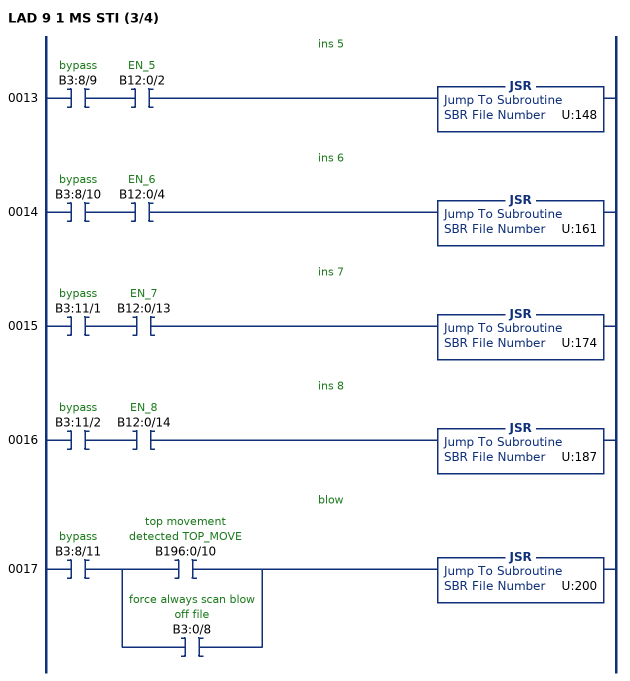
% Rung: 13 %
% ins 5 %
SOR XIC B3:8/9 XIC B12:0/2 JSR U:148 EOR
%   B3:8/9  "bypass" %
%   B12:0/2  EN_5 %
% Rung: 14 %
% ins 6 %
SOR XIC B3:8/10 XIC B12:0/4 JSR U:161 EOR
%   B3:8/10  "bypass" %
%   B12:0/4  EN_6 %
% Rung: 15 %
% ins 7 %
SOR XIC B3:11/1 XIC B12:0/13 JSR U:174 EOR
%   B3:11/1  "bypass" %
%   B12:0/13  EN_7 %
% Rung: 16 %
% ins 8 %
SOR XIC B3:11/2 XIC B12:0/14 JSR U:187 EOR
%   B3:11/2  "bypass" %
%   B12:0/14  EN_8 %
% Rung: 17 %
% blow %
SOR XIC B3:8/11 BST XIC B196:0/10 NXB XIC B3:0/8 BND JSR U:200 EOR
%   B3:8/11  "bypass" %
%   B196:0/10  TOP_MOVE  "top movement detected" %
%   B3:0/8  "force always scan blow off file" %

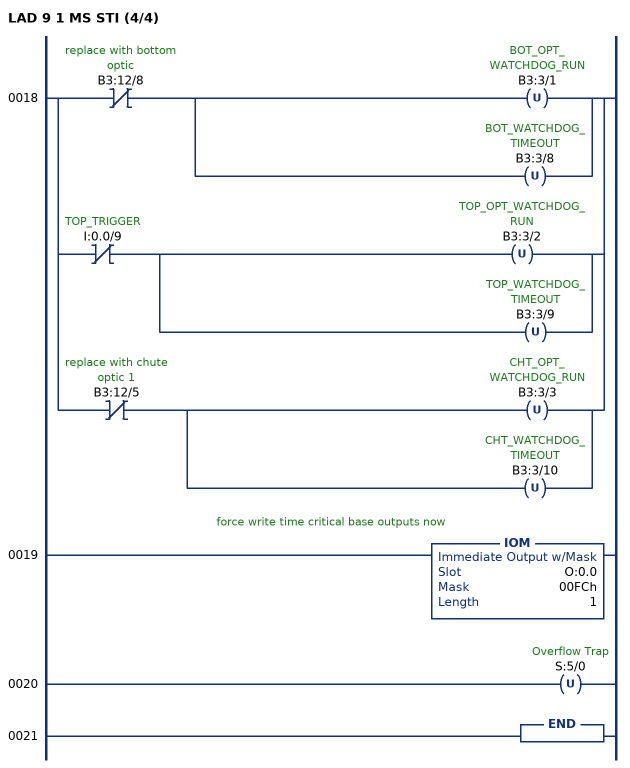
% Rung: 18 %
SOR BST XIO B3:12/8 BST OTU B3:3/1 NXB OTU B3:3/8 BND NXB XIO I:0.0/9 BST OTU B3:3/2 NXB OTU B3:3/9 BND NXB XIO B3:12/5 BST OTU B3:3/3 NXB OTU B3:3/10 BND BND EOR
%   B3:12/8  "replace with bottom optic" %
%   B3:3/1  BOT_OPT_WATCHDOG_RUN %
%   B3:3/8  BOT_WATCHDOG_TIMEOUT %
%   I:0.0/9  TOP_TRIGGER %
%   B3:3/2  TOP_OPT_WATCHDOG_RUN %
%   B3:3/9  TOP_WATCHDOG_TIMEOUT %
%   B3:12/5  "replace with chute optic 1" %
%   B3:3/3  CHT_OPT_WATCHDOG_RUN %
%   B3:3/10  CHT_WATCHDOG_TIMEOUT %
% Rung: 19 %
% force write time critical base outputs now %
SOR IOM O:0.0 00FCh 1 EOR
% Rung: 20 %
SOR OTU S:5/0 EOR
%   S:5/0  "Overflow Trap" %
% Rung: 21 %
SOR END EOR

LADDER 10 "SHIFT BOT"
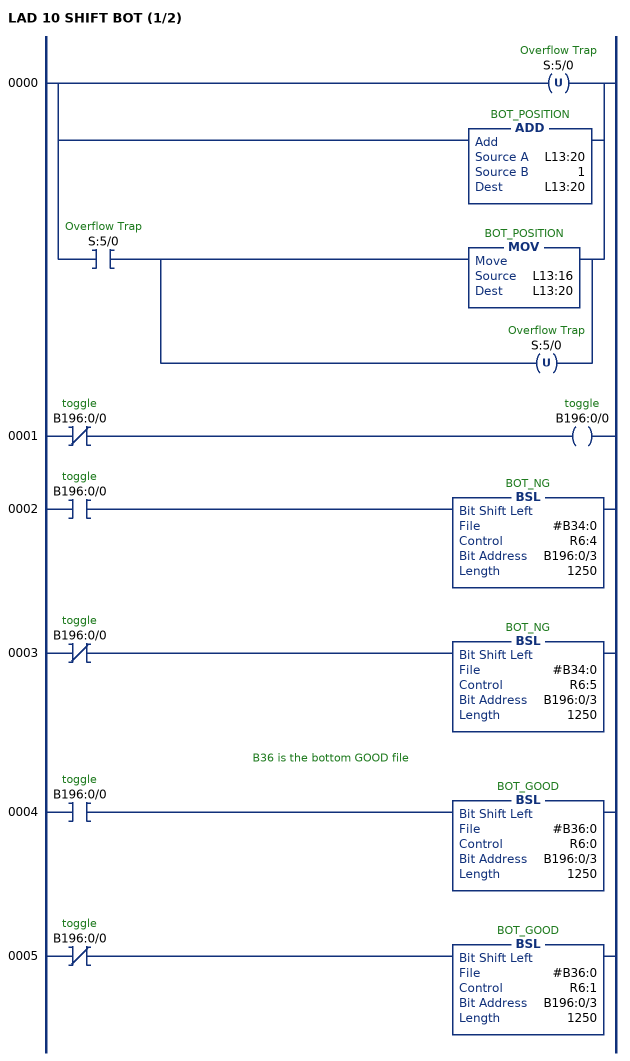
% Rung: 0 %
SOR BST OTU S:5/0 NXB ADD L13:20 1 L13:20 NXB XIC S:5/0 BST MOV L13:16 L13:20 NXB OTU S:5/0 BND BND EOR
%   S:5/0  "Overflow Trap" %
%   L13:20  BOT_POSITION %
%   L13:16  MIN_LONG %
% Rung: 1 %
SOR XIO B196:0/0 OTE B196:0/0 EOR
%   B196:0/0  "toggle" %
% Rung: 2 %
SOR XIC B196:0/0 BSL #B34:0 R6:4 B196:0/3 1250 EOR
%   B196:0/0  "toggle" %
%   B34:0  BOT_NG %
%   B196:0/3  OFF %
% Rung: 3 %
SOR XIO B196:0/0 BSL #B34:0 R6:5 B196:0/3 1250 EOR
%   B196:0/0  "toggle" %
%   B34:0  BOT_NG %
%   B196:0/3  OFF %
% Rung: 4 %
% B36 is the bottom GOOD file %
SOR XIC B196:0/0 BSL #B36:0 R6:0 B196:0/3 1250 EOR
%   B196:0/0  "toggle" %
%   B36:0  BOT_GOOD %
%   B196:0/3  OFF %
% Rung: 5 %
SOR XIO B196:0/0 BSL #B36:0 R6:1 B196:0/3 1250 EOR
%   B196:0/0  "toggle" %
%   B36:0  BOT_GOOD %
%   B196:0/3  OFF %

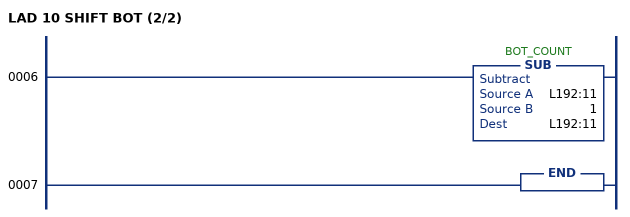
% Rung: 6 %
SOR SUB L192:11 1 L192:11 EOR
%   L192:11  BOT_COUNT %
% Rung: 7 %
SOR END EOR

LADDER 11 "SHIFT TOP"
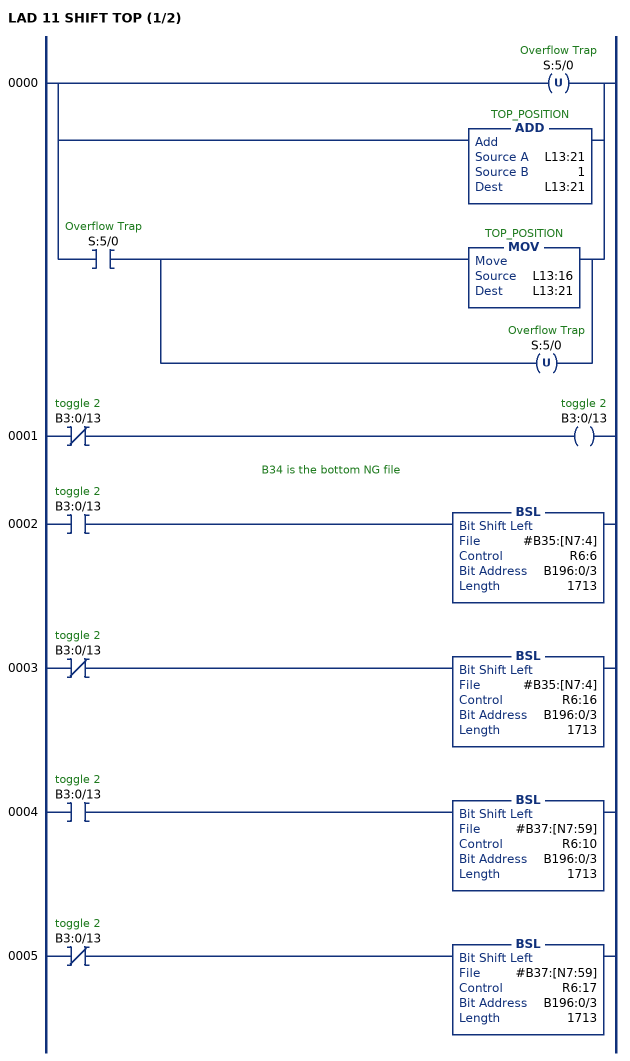
% Rung: 0 %
SOR BST OTU S:5/0 NXB ADD L13:21 1 L13:21 NXB XIC S:5/0 BST MOV L13:16 L13:21 NXB OTU S:5/0 BND BND EOR
%   S:5/0  "Overflow Trap" %
%   L13:21  TOP_POSITION %
%   L13:16  MIN_LONG %
% Rung: 1 %
SOR XIO B3:0/13 OTE B3:0/13 EOR
%   B3:0/13  "toggle 2" %
% Rung: 2 %
% B34 is the bottom NG file %
SOR XIC B3:0/13 BSL #B35:[N7:4] R6:6 B196:0/3 1713 EOR
%   B3:0/13  "toggle 2" %
%   N7:4  TOP_NG_START_WORD %
%   B196:0/3  OFF %
% Rung: 3 %
SOR XIO B3:0/13 BSL #B35:[N7:4] R6:16 B196:0/3 1713 EOR
%   B3:0/13  "toggle 2" %
%   N7:4  TOP_NG_START_WORD %
%   B196:0/3  OFF %
% Rung: 4 %
SOR XIC B3:0/13 BSL #B37:[N7:59] R6:10 B196:0/3 1713 EOR
%   B3:0/13  "toggle 2" %
%   N7:59  TOP_GOOD1_START_WORD %
%   B196:0/3  OFF %
% Rung: 5 %
SOR XIO B3:0/13 BSL #B37:[N7:59] R6:17 B196:0/3 1713 EOR
%   B3:0/13  "toggle 2" %
%   N7:59  TOP_GOOD1_START_WORD %
%   B196:0/3  OFF %

